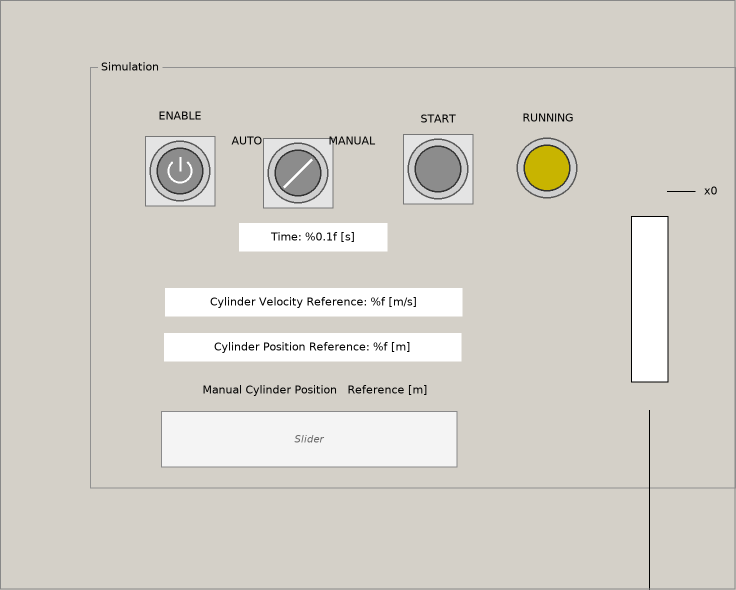
VISUALIZATION CraneHMI  // 736x590
    Rectangle (566,281 166x37), angle 270
    GroupBox (90,59 646x429), "Simulation"
        PowerSwitch (55,77 70x70), variable: Inputs.bEnableSimulation, behaviour: TOGGLE, style: Switch-PowerSwitch-Gray
        PushSwitch (313,75 70x70), variable: Inputs.bStartSimulation, behaviour: TOGGLE, style: Switch-PushSwitch-Gray
        Lamp1 (422,74 70x70), variable: Outputs.bSimulationRunning, style: Lamp-Lamp1-Yellow
        Textfield (74,228 299x30), "Cylinder Velocity Reference: %f [m/s]", text variable: Inputs.fCylinderVelocityReference
            OnMouseClick: write the text variable via Default
        Label (15,42 150x30), "ENABLE"
        Label (273,45 150x30), "START"
        Label (383,44 150x30), "RUNNING"
        Textfield (148,163 150x30), "Time: %0.1f [s]", text variable: Outputs.fSimulationTime
        Slider (71,352 296x56), variable: Inputs.fManualCylinderPositionReference, scale 0..1
        RotarySwitch (173,79 70x70), variable: Inputs.bAutoMode, behaviour: TOGGLE, style: Switch-RotarySwitch-Gray
        Label (82,67 150x30), "AUTO"
        Label (187,67 150x30), "MANUAL"
        Label (90,316 270x30), "Manual Cylinder Position Reference [m]"
        Textfield (73,273 299x30), "Cylinder Position Reference: %f [m]", text variable: Inputs.fManualCylinderPositionReference
        Line (577,132) (605,132)
        Label (607,117 28x30), "x0"
    Line (649,410) (649,590)
        p1126004900: Outputs.pt1_y
        p3528305787: Outputs.pt0_x
        p2773130477: Outputs.pt0_y
        p874137650: Outputs.pt1_x
    Line (706,188) (706,188)
END_VISUALIZATION

(* stored: Version 1.1.0.1, ProductVersion 3.1.4024.10
   Visu CraneHMI: Id {4bdd8ed7-7379-4dd1-955f-a8a1c50d5ff4} *)
